TYPE ST_RemoteCtrlSection EXTENDS ST_SectionBase :
STRUCT
END_STRUCT
END_TYPE

(* stored: Version 1.1.0.1, ProductVersion 3.1.4024.12
   DUT ST_RemoteCtrlSection: Id {9f2d6d22-e9a9-4f6c-992a-961c2c122615} *)
